Staubli VAL3: onExit.pgx

program onExit(bool& x_bSave[])
  local string l_sMessage
  local bool l_bYes
  local frame l_fNewWorld
  local bool l_bCancel
  local string l_sButton[2]
  local num l_nResult
begin
//  // saveIt
//  if x_bSave
//    call language:message(l_sMessage,-1)
//    // get the yes_no button
//    call language:getYesNo(l_sButton)
//    // ask the question
//    call use:yes_no_cancel(l_sMessage,l_sButton,l_bYes,l_bCancel)
//    if l_bYes
//      call saveIt(x_bSave)
//    else
//      sItems[0]=""
//    endIf
//    // look for the cancel button to cancel
//    bExit=!l_bCancel
//  else
//    // exit from the page
//    bExit=true
//  endIf
//  // resetMotion
//  if !cycleStatus:bCycle
//    resetMotion()
//  endIf
//  // give back
//  // set the number
//  if size(sItems)>1
//    sItems[1]=toString("",nSelect)
//  endIf
//  // reset the show status
//  bShowStatus=false
//  //
//  call tcp:getTool(tTool,saveData:nIndexTool)
//  // give back the jog context
//  saveData:nFrameActive=nBackupFrame
//  fFather=saveData:fFrameItem[saveData:nFrameActive].fFrame
//  $jogContext(tTool,fFather,0)
end
